TYPE DeviceDataEval :
STRUCT
	
	OEM: STRING(50);
	OMEModelName: STRING(50);
	OEMModelCode: STRING(50);
	Model: STRING(50);
	Color: STRING(50);
	OSName: STRING(50);
	OSVersion: STRING(50);
	Profile: STRING(50);
	Carrier: STRING(50);
	IMEI: STRING(30);

END_STRUCT
END_TYPE

(* stored: Version 1.1.0.1, ProductVersion 3.1.4024.6
   DUT DeviceDataEval: Id {afa32f1c-e3ba-459e-92e6-b2f04f6205ab} *)
